{attribute 'linkalways'} 
{attribute 'no_explicit_call' := 'This FB is a CLASS and must be accessed using methods or properties'}
{attribute 'enable_dynamic_creation'}
FUNCTION_BLOCK Node_F_VN_AppendToContainer_LREAL EXTENDS VisionNode
VAR
    fElement : _LREAL(0.0);
    ipContainer : _ITcVnContainer;
    hrPrev : _HRESULT(S_OK);
	hresult : _HRESULT(S_OK);
END_VAR

METHOD PUBLIC  Clone : I_Node
VAR
	pNode : POINTER TO Node_F_VN_AppendToContainer_LREAL;
END_VAR
pNode := __NEW(Node_F_VN_AppendToContainer_LREAL);
Clone := pNode^;
END_METHOD

METHOD FB_init : BOOL
VAR_INPUT
	bInitRetains : BOOL; // if TRUE, the retain variables are initialized (warm start / cold start)
	bInCopyCode : BOOL;  // if TRUE, the instance afterwards gets moved into the copy code (online change)
END_VAR
AddInput('fElement', fElement);
AddInput('ipContainer', ipContainer);
AddInput('hrPrev', hrPrev);
AddOutput('ipContainer', ipContainer);
AddOutput('hresult',hresult);
END_METHOD

METHOD PROTECTED OnExecute : HRESULT
hresult.Value := F_VN_AppendToContainer_LREAL(
    fElement := fElement.Value,
	ipContainer := ipContainer.Value,
	hrPrev:= hrPrev.Value);
END_METHOD

METHOD PUBLIC PreExecutionCheck
VAR_INPUT
	Check : I_PreExecutionChecks;
END_VAR
Check.IsTrue(ipContainer.IsValid, 'ipContainer must be a valid container');
Check.IsTrue(ipContainer.HasType('CTcVnContainer_Vector_LREAL'), 'ipContainer contains incorrect types');
END_METHOD

END_FUNCTION_BLOCK

(* stored: Version 1.1.0.1, ProductVersion 3.1.4024.13
   POU Node_F_VN_AppendToContainer_LREAL: Id {9c456dd0-8fbf-0f09-330d-256acff0954a}, SpecialFunc None
   Folder Constructor: Id {dc0ee5f1-f0ae-04ec-15c9-08fa8099b305}
   Method Clone: Id {cfd72875-b6bf-01da-0e29-ea30225aa61d}
   Method FB_init: Id {d1fdff74-f2ce-0765-1e05-e50609f007e4}
   Method OnExecute: Id {645d6e30-a2f9-0d05-1666-f72cda26670a}
   Method PreExecutionCheck: Id {b2cc5b62-217d-0e17-2f9c-50e1c29bf83b} *)
